// TIA Portal V19 export
DATA_BLOCK "instU1ConstraintTray"   // DB8
AUTHOR : SUP/Zhang Shi Long
FAMILY : SUP
// stored: InstanceOfName LEXCHANGETRAY_UpdateMaterialInfo, InstanceOfType FB
"LEXCHANGETRAY_UpdateMaterialInfo"
   // VAR_IN_OUT
   //    materialInterface : "LEXCHANGETRAY_typeTrayInterface";
   // END_VAR
   // VAR
   //    lstPostion : "LEXCHANGETRAY_typeTrayPosition";
   //    I { S7_SetPoint := 'True'} : Int;
   //    upperBound : Int;
   // END_VAR
BEGIN
END_DATA_BLOCK
